FUNCTION IsNaN : BOOL
VAR_INPUT
	IN : REAL;
END_VAR
VAR
	tempdword : DWORD;
	testword : WORD;
END_VAR

tempdword := PDWORD_TO_DWORD(ADR(In));
memcpy(ADR(TestWord), ADR(tempdword) +2, 2);

IsNaN := ((TestWord AND 2#0111111110000000) = 2#0111111110000000);

END_FUNCTION

(* stored: Version 1.1.0.1, ProductVersion 3.1.4026.18
   POU IsNaN: Id {93707678-1d3c-43be-907f-47bf14dc034d}, SpecialFunc None *)
